FUNCTION_BLOCK Delay
VAR_INPUT
	Delay_On	: BOOL;
	Delay_Time	: TIME;
END_VAR
VAR_OUTPUT
	Delay_Done	: BOOL;
END_VAR

END_FUNCTION_BLOCK

(* stored: Version 1.1.0.1, ProductVersion 3.1.4020.12
   POU Delay: Id {9b91272d-9848-4c41-8af9-1af6a2bdd545}, SpecialFunc None *)
